Universal Robots PolyScope program: Pallet1.0_PF.urp

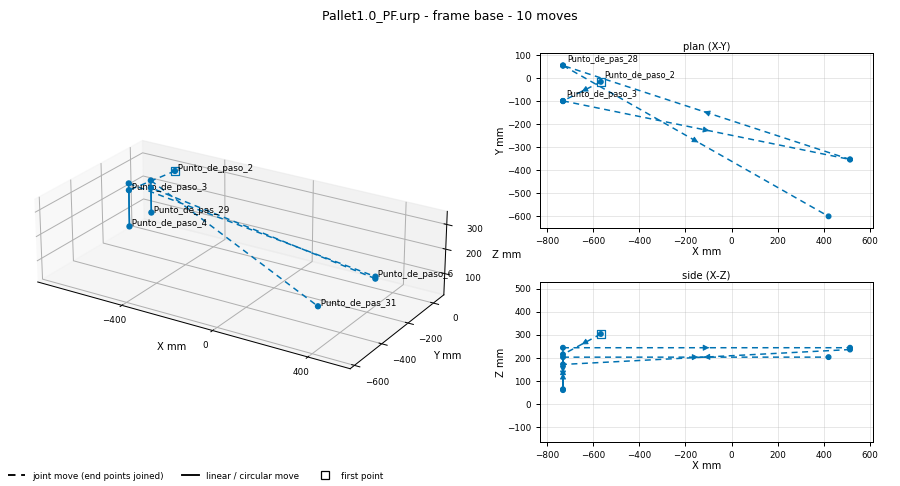
[picture p0: tool path of Pallet1.0_PF.urp in frame base, 10 of 10 moves have a stored position in this frame; points joined in program order, loops and branches not executed]
Program Pallet1.0_PF (installation=default directory=/programs/usbdisk_0 createdIn=3.15.8.106339 lastSavedIn=3.15.8.106339 robotSerialNumber=2015350901)
Calibrated DH parameters: a=[0, -0.425, -0.39225, 0, 0, 0]; d=[0.089159, 0, 0, 0.10915, 0.09465, 0.0823]; alpha=[1.570796, 0, 0, 1.570796, -1.570796, 0]; deltaTheta=[0, 0, 0, 0, 0, 0]
Robot Program (runOnlyOnce=false)
  MoveJ speed 60 deg/s, acceleration 80 deg/s^2 (useActiveTCP=true)
    Waypoint Punto_de_paso_2: TCP in base x=-566.321 y=-16.438 z=304.18 mm, rx=2.2273 ry=2.2091 rz=0.0057 rad; joints [-9.438, -79.943, 72.118, -81.838, -90.015, -8.968] deg; flange x=-567.338 y=-16.315 z=478.176 mm, rx=2.2273 ry=2.2091 rz=0.0057 rad
    If digital_in[1]≟ True
      MoveJ speed 60 deg/s, acceleration 80 deg/s^2 (useActiveTCP=true)
        Waypoint Punto_de_paso_3: TCP in base x=-730.444 y=-98.928 z=215.761 mm, rx=2.2274 ry=2.209 rz=0.0055 rad; joints [-0.817, -54.762, 49.45, -84.36, -89.96, -0.342] deg; flange x=-731.439 y=-98.792 z=389.758 mm, rx=2.2274 ry=2.209 rz=0.0055 rad
        MoveL speed 250 mm/s, acceleration 1200 mm/s^2 (useActiveTCP=true) feature=Base
          Waypoint Punto_de_paso_4: TCP in base x=-730.393 y=-100.609 z=60.935 mm, rx=2.2272 ry=2.209 rz=0.0056 rad; joints [-0.686, -52.453, 68.486, -105.697, -89.955, -0.217] deg; flange x=-731.413 y=-100.461 z=234.932 mm, rx=2.2272 ry=2.209 rz=0.0056 rad
          URCap Gripper (Robotiq_Grippers, Robotiq Inc.) dataModel(position=100.0, force=100.0, speed=100.0, positionInDouble=100.0, forceInDouble=100.0, speedInDouble=100.0, slaveIds=[9], blocking=true); state(isChildrenLocked=true)
          Waypoint Punto_de_paso_5: TCP in base x=-730.487 y=-98.949 z=244.682 mm, rx=2.2273 ry=2.2091 rz=0.0053 rad; joints [-0.817, -54.045, 44.014, -79.647, -89.955, -0.345] deg; flange x=-731.462 y=-98.799 z=418.679 mm, rx=2.2273 ry=2.2091 rz=0.0053 rad
          MoveJ speed 60 deg/s, acceleration 80 deg/s^2 (useActiveTCP=true)
            Waypoint Punto_de_paso_6: TCP in base x=513.312 y=-352.994 z=244.725 mm, rx=2.2039 ry=-2.2386 rz=-0.0089 rad; joints [135.397, -72.477, 71.437, -88.635, -90.007, -43.708] deg; flange x=514.03 y=-353.672 z=418.722 mm, rx=2.2039 ry=-2.2386 rz=-0.0089 rad
          MoveL speed 250 mm/s, acceleration 1200 mm/s^2 (useActiveTCP=true) feature=Base
            Waypoint Punto_de_paso_7: TCP in base x=513.278 y=-353.004 z=236.797 mm, rx=2.2038 ry=-2.2387 rz=-0.0091 rad; joints [135.393, -72.485, 72.603, -89.786, -90.006, -43.706] deg; flange x=514.01 y=-353.701 z=410.794 mm, rx=2.2038 ry=-2.2387 rz=-0.0091 rad
            Pallet pattern(dimensionality=List firstAxisCount=5 secondAxisCount=5 thirdAxisCount=5 motionType=MoveL speed=0.25 acceleration=1.2 useActiveTCP=true, counterVariable(name=cont_1, initializeExpression=0), patternPoseVariable(name=pose_1), feature=Base, children(Waypoint(type=Fixed name=Punto_de_paso_8, position(joints=2.3631303310394287, -1.1275900045977991, 1.6604909896850586, -2.0977628866778772, -1.571042839680807, -0.7629154364215296 pose=0.5132245674611735, -0.3529411145356251, 0.01696247469393014, 2.203863236658737, -2.2383939411612848, -0.009314066402786586), poseInFeatureCoordinates=[0.513225, -0.352941, 0.016962, 2.203863, -2.238394, -0.009314], outputFlangePose=[0.51399, -0.353636, 0.190959, 2.203863, -2.238394, -0.009314]), Waypoint(type=Fixed name=Punto_de_paso_9, position(joints=2.4081342220306396, -1.0566390196429651, 1.545675277709961, -2.05412465730776, -1.570719067250387, -0.7178614775287073 pose=0.5548105961057649, -0.3530178817913074, 0.018104225127487772, 2.2038560559889255, -2.2385008669096638, -0.008956480055837733), poseInFeatureCoordinates=[0.554811, -0.353018, 0.018104, 2.203856, -2.238501, -0.008956], outputFlangePose=[0.555539, -0.353693, 0.192101, 2.203856, -2.238501, -0.008956]), Waypoint(type=Fixed name=Punto_de_pas_10, position(joints=2.446105718612671, -0.9861076513873499, 1.4307241439819336, -2.0095513502704065, -1.5704076925860804, -0.6796610991107386 pose=0.5934753632034022, -0.35301619621523517, 0.017998009023001, 2.203652981289238, -2.2388090833039787, -0.009222219608768033), poseInFeatureCoordinates=[0.593475, -0.353016, 0.017998, 2.203653, -2.238809, -0.009222], outputFlangePose=[0.594215, -0.353722, 0.191995, 2.203653, -2.238809, -0.009222]), Waypoint(type=Fixed name=Punto_de_pas_11, position(joints=2.480747699737549, -0.9116233030902308, 1.3046913146972656, -1.958066765462057, -1.5702398459063929, -0.6444733778582972 pose=0.6321841473893125, -0.35306041061215476, 0.018035419146744114, 2.20302057784513, -2.2393896017985955, -0.009141742887616903), poseInFeatureCoordinates=[0.632184, -0.35306, 0.018035, 2.203021, -2.23939, -0.009142], outputFlangePose=[0.632921, -0.353756, 0.192032, 2.203021, -2.23939, -0.009142]), Waypoint(type=Fixed name=Punto_de_pas_12, position(joints=2.515030860900879, -0.8245127836810511, 1.1525378227233887, -1.892914120350973, -1.570024315510885, -0.6107981840716761 pose=0.6740908514581094, -0.3529593660500304, 0.017973942492954004, 2.2036977466389036, -2.238717787266496, -0.00935099502202368), poseInFeatureCoordinates=[0.674091, -0.352959, 0.017974, 2.203698, -2.238718, -0.009351], outputFlangePose=[0.674845, -0.353671, 0.191971, 2.203698, -2.238718, -0.009351]), Waypoint(type=Fixed name=Punto_de_pas_13, position(joints=2.3630945682525635, -1.169779125844137, 1.6140356063842773, -2.009144131337301, -1.5711506048785608, -0.7630236784564417 pose=0.5131685944157, -0.35295550636586853, 0.05500279295848928, 2.2038697585970315, -2.2382376084810494, -0.00927087314573258), poseInFeatureCoordinates=[0.513169, -0.352956, 0.055003, 2.20387, -2.238238, -0.009271], outputFlangePose=[0.513944, -0.353634, 0.229, 2.20387, -2.238238, -0.009271]), Waypoint(type=Fixed name=Punto_de_pas_14, position(joints=2.4080862998962402, -1.094360653554098, 1.500410556793213, -1.9713957945453089, -1.5707791487323206, -0.7179215590106409 pose=0.5548164047230572, -0.35308568147939057, 0.05508461053102831, 2.20383957497247, -2.23845651633265, -0.008547041026006829), poseInFeatureCoordinates=[0.554816, -0.353086, 0.055085, 2.20384, -2.238457, -0.008547], outputFlangePose=[0.555519, -0.353723, 0.229082, 2.20384, -2.238457, -0.008547]), Waypoint(type=Fixed name=Punto_de_pas_15, position(joints=2.446117877960205, -1.021660629902975, 1.383436679840088, -1.9266999403582972, -1.570467774068014, -0.6796610991107386 pose=0.5934677735696893, -0.35301912054014967, 0.0559910473342225, 2.2036240498734854, -2.238752074764261, -0.00922996533762203), poseInFeatureCoordinates=[0.593468, -0.353019, 0.055991, 2.203624, -2.238752, -0.00923], outputFlangePose=[0.594216, -0.353718, 0.229988, 2.203624, -2.238752, -0.00923]), Waypoint(type=Fixed name=Punto_de_pas_16, position(joints=2.480783700942993, -0.9441817442523401, 1.2555980682373047, -1.8764341513263147, -1.5702040831195276, -0.6444852987872522 pose=0.6321844252540715, -0.3530163761280898, 0.05638557463513269, 2.203100752356905, -2.2393639874148366, -0.009119588993108625), poseInFeatureCoordinates=[0.632184, -0.353016, 0.056386, 2.203101, -2.239364, -0.00912], outputFlangePose=[0.632915, -0.353715, 0.230383, 2.203101, -2.239364, -0.00912]), Waypoint(type=Fixed name=Punto_de_pas_17, position(joints=2.515138626098633, -0.8528311888324183, 1.1003336906433105, -1.8122723738299769, -1.5700843969928187, -0.6107738653766077 pose=0.6741036541561095, -0.35288746982087266, 0.05628562580244548, 2.2037352226759186, -2.238568724907899, -0.009519706762820677), poseInFeatureCoordinates=[0.674104, -0.352887, 0.056286, 2.203735, -2.238569, -0.00952], outputFlangePose=[0.674881, -0.353603, 0.230282, 2.203735, -2.238569, -0.00952]), Waypoint(type=Fixed name=Punto_de_pas_18, position(joints=2.363046646118164, -1.2044346968280237, 1.5590686798095703, -1.9196580092059534, -1.5711386839496058, -0.7629631201373499 pose=0.5131860409950756, -0.3530097003409165, 0.09290491266257156, 2.203758462356244, -2.2383675429672354, -0.009057018848740528), poseInFeatureCoordinates=[0.513186, -0.35301, 0.092905, 2.203758, -2.238368, -0.009057], outputFlangePose=[0.513943, -0.353673, 0.266902, 2.203758, -2.238368, -0.009057]), Waypoint(type=Fixed name=Punto_de_pas_19, position(joints=2.408074378967285, -1.1262005011187952, 1.4451117515563965, -1.8843262831317347, -1.5708149115191858, -0.7178857962237757 pose=0.5548151996713835, -0.3531073422909641, 0.0930535390031054, 2.2037643292926323, -2.2384866218002153, -0.008435196605507001), poseInFeatureCoordinates=[0.554815, -0.353107, 0.093054, 2.203764, -2.238487, -0.008435], outputFlangePose=[0.555513, -0.353732, 0.267051, 2.203764, -2.238487, -0.008435]), Waypoint(type=Fixed name=Punto_de_pas_20, position(joints=2.446141481399536, -1.049763027821676, 1.3284411430358887, -1.8438447157489222, -1.5705392996417444, -0.6796248594867151 pose=0.593499660509277, -0.3530486469996806, 0.09303287538988136, 2.20357754039206, -2.238732576216275, -0.008839450693340935), poseInFeatureCoordinates=[0.5935, -0.353049, 0.093033, 2.203578, -2.238733, -0.008839], outputFlangePose=[0.594223, -0.353711, 0.26703, 2.203578, -2.238733, -0.008839]), Waypoint(type=Fixed name=Punto_de_pas_21, position(joints=2.4808316230773926, -0.9693010489093226, 1.1972637176513672, -1.792868439351217, -1.5702760855304163, -0.6445453802691858 pose=0.6321624175986366, -0.35297919711606884, 0.09406846161006818, 2.20316112021239, -2.2391830633267427, -0.009278826783431064), poseInFeatureCoordinates=[0.632162, -0.352979, 0.094068, 2.203161, -2.239183, -0.009279], outputFlangePose=[0.632916, -0.35368, 0.268065, 2.203161, -2.239183, -0.009279]), Waypoint(type=Fixed name=Punto_de_pas_22, position(joints=2.5151865482330322, -0.8737342993365687, 1.0374155044555664, -1.7285955587970179, -1.570144001637594, -0.6108344236956995 pose=0.674108251554734, -0.3528651117998487, 0.09425003366463722, 2.2038330133524338, -2.2384246855338255, -0.009280286167645216), poseInFeatureCoordinates=[0.674108, -0.352865, 0.09425, 2.203833, -2.238425, -0.00928], outputFlangePose=[0.674871, -0.353557, 0.268247, 2.203833, -2.238425, -0.00928]), Waypoint(type=Fixed name=Punto_de_pas_23, position(joints=2.3629984855651855, -1.2317708174334925, 1.4950027465820312, -1.8283217589007776, -1.571174446736471, -0.7630112806903284 pose=0.5131707080842348, -0.35304893689303485, 0.1310672998062101, 2.2037345545345137, -2.238343056471053, -0.008952794505665341), poseInFeatureCoordinates=[0.513171, -0.353049, 0.131067, 2.203735, -2.238343, -0.008953], outputFlangePose=[0.513924, -0.353699, 0.305064, 2.203735, -2.238343, -0.008953]), Waypoint(type=Fixed name=Punto_de_pas_24, position(joints=2.408074378967285, -1.1507447401629847, 1.3807148933410645, -1.7955272833453577, -1.5708630720721644, -0.7178013960467737 pose=0.554819388099037, -0.35312773426757993, 0.13100770525803954, 2.203642492159454, -2.238551534923004, -0.00820777086849384), poseInFeatureCoordinates=[0.554819, -0.353128, 0.131008, 2.203642, -2.238552, -0.008208], outputFlangePose=[0.555504, -0.353729, 0.305005, 2.203642, -2.238552, -0.008208]), Waypoint(type=Fixed name=Punto_de_pas_25, position(joints=2.445997953414917, -1.0713494459735315, 1.2620959281921387, -1.7558816115008753, -1.5705512205706995, -0.6796129385577601 pose=0.5934510057003118, -0.353139496484484, 0.1310450990567559, 2.2033932515905694, -2.2388933313548534, -0.008886805674271178), poseInFeatureCoordinates=[0.593451, -0.353139, 0.131045, 2.203393, -2.238893, -0.008887], outputFlangePose=[0.59418, -0.353803, 0.305042, 2.203393, -2.238893, -0.008887]), Waypoint(type=Fixed name=Punto_de_pas_26, position(joints=2.480879545211792, -0.9869101683246058, 1.1285271644592285, -1.7065790335284632, -1.5703237692462366, -0.6446173826800745 pose=0.6321941557152236, -0.3529759022987843, 0.13153622061743322, 2.2032678780951342, -2.2390226574753136, -0.009181205365187293), poseInFeatureCoordinates=[0.632194, -0.352976, 0.131536, 2.203268, -2.239023, -0.009181], outputFlangePose=[0.632945, -0.353664, 0.305533, 2.203268, -2.239023, -0.009181]), Waypoint(type=Fixed name=Punto_de_pas_27, position(joints=2.5152344703674316, -0.8862040678607386, 0.9623470306396484, -1.6410678068744105, -1.5702160040484827, -0.6108582655536097 pose=0.6741341209130111, -0.35286206802645803, 0.13170720668516567, 2.203865000162463, -2.238296039311312, -0.009245053414911254), poseInFeatureCoordinates=[0.674134, -0.352862, 0.131707, 2.203865, -2.238296, -0.009245], outputFlangePose=[0.674903, -0.353543, 0.305704, 2.203865, -2.238296, -0.009245]))); actionSequence(name=SecuenciaPalé motionType=MoveL speed=0.25 acceleration=1.2 useActiveTCP=true, anchorWaypoint(type=Fixed name=PuntoDePatrón_1, position(joints=2.3631303310394287, -1.1276257673846644, 1.6605868339538574, -2.097715202962057, -1.5710185209857386, -0.7629755179034632 pose=0.5131909342788984, -0.35289919057667213, 0.01693865784924231, 2.2039461302595416, -2.238343765061751, -0.00948395217768327), poseInFeatureCoordinates=[0.513191, -0.352899, 0.016939, 2.203946, -2.238344, -0.009484], outputFlangePose=[0.513967, -0.35361, 0.190935, 2.203946, -2.238344, -0.009484]), feature=Base, children(Waypoint(type=Fixed name=Acercar_1, position(joints=2.3878726959228516, -1.1627238432513636, 1.499763011932373, -1.901944939290182, -1.5708869139300745, -0.738204304371969 pose=0.535486537471644, -0.35292770718209365, 0.09269323575355731, 2.2039055569885972, -2.238368044698761, -0.009239097655524674), poseInFeatureCoordinates=[0.535487, -0.352928, 0.092693, 2.203906, -2.238368, -0.009239], outputFlangePose=[0.536245, -0.353618, 0.26669, 2.203906, -2.238368, -0.009239]), Waypoint=PuntoDePatrón_1, Contributed(strategyProgramNodeType=Gripper strategyURCapDeveloper=Robotiq Inc. strategyURCapName=Robotiq_Grippers, dataModel(position=0.0, force=100.0, speed=100.0, positionInDouble=0.0, forceInDouble=100.0, speedInDouble=100.0, slaveIds=[9], blocking=true), state(isChildrenLocked=true)), Set(type=NoAction), Wait(type=Sleep, waitTime=1), Waypoint(type=Fixed name=Salir_1, position(joints=2.3556182384490967, -1.2753384749041956, 1.433816909790039, -1.7237561384784144, -1.5711506048785608, -0.7702725569354456 pose=0.5042328769515484, -0.35049239066438986, 0.17702159380140353, 2.2036488263975693, -2.2385225445096353, -0.008663256964435576), poseInFeatureCoordinates=[0.504233, -0.350492, 0.177022, 2.203649, -2.238523, -0.008663], outputFlangePose=[0.504955, -0.351128, 0.351019, 2.203649, -2.238523, -0.008663])))
              Pattern -> pattern
              AnchoredSequence -> SecuenciaPalé
    ElseIf digital_in[0]≟ True
      MoveJ speed 60 deg/s, acceleration 80 deg/s^2 (useActiveTCP=true)
        Waypoint Punto_de_pas_28: TCP in base x=-730.325 y=54.404 z=172.261 mm, rx=2.2271 ry=2.2089 rz=0.0058 rad; joints [-12.82, -55.781, 57.455, -91.329, -90.032, -12.349] deg; flange x=-731.369 y=54.543 z=346.257 mm, rx=2.2271 ry=2.2089 rz=0.0058 rad
        MoveL speed 250 mm/s, acceleration 1200 mm/s^2 (useActiveTCP=true) feature=Base
          Waypoint Punto_de_pas_29: TCP in base x=-730.375 y=54.354 z=64.707 mm, rx=2.2272 ry=2.2093 rz=0.0057 rad; joints [-12.814, -53.288, 69.317, -105.701, -90.036, -12.35] deg; flange x=-731.373 y=54.469 z=238.705 mm, rx=2.2272 ry=2.2093 rz=0.0057 rad
          URCap Gripper (Robotiq_Grippers, Robotiq Inc.) dataModel(position=100.0, force=100.0, speed=100.0, positionInDouble=100.0, forceInDouble=100.0, speedInDouble=100.0, slaveIds=[9], blocking=true); state(isChildrenLocked=true)
          Waypoint Punto_de_pas_30: TCP in base x=-730.317 y=54.385 z=203.798 mm, rx=2.2271 ry=2.209 rz=0.0058 rad; joints [-12.819, -55.724, 52.756, -86.687, -90.032, -12.352] deg; flange x=-731.359 y=54.522 z=377.794 mm, rx=2.2271 ry=2.209 rz=0.0058 rad
          MoveJ speed 60 deg/s, acceleration 80 deg/s^2 (useActiveTCP=true)
            Waypoint Punto_de_pas_31: TCP in base x=420.29 y=-599.707 z=203.949 mm, rx=-2.196 ry=2.245 rz=0.009 rad; joints [116.465, -55.735, 52.753, -86.686, -90.037, -62.27] deg; flange x=420.842 y=-600.562 z=377.946 mm, rx=-2.196 ry=2.245 rz=0.009 rad
            Pallet pattern(dimensionality=List firstAxisCount=5 secondAxisCount=5 thirdAxisCount=5 motionType=MoveL speed=0.25 acceleration=1.2 useActiveTCP=true, counterVariable(name=cont_2, initializeExpression=0), patternPoseVariable(name=pose_2), feature=Base, children(Waypoint(type=Fixed name=Punto_de_pas_32, position(joints=2.0326786041259766, -0.9004228750811976, 1.2612924575805664, -1.9260895887957972, -1.5714500586139124, -1.0868600050555628 pose=0.42031223679203245, -0.5997915862684211, 0.026862123093794543, -2.1960409743045224, 2.245010484936809, 0.008647737661910772), poseInFeatureCoordinates=[0.420312, -0.599792, 0.026862, -2.196041, 2.24501, 0.008648], outputFlangePose=[0.420846, -0.60061, 0.200859, -2.196041, 2.24501, 0.008648]), Waypoint(type=Fixed name=Punto_de_pas_33, position(joints=1.9777237176895142, -0.952315632496969, 1.3581628799438477, -1.9710243383990687, -1.5718210379229944, -1.1419809500323694 pose=0.377052081475406, -0.59975092745355, 0.023745193947307175, -2.1962488525573267, 2.2448477292954836, 0.00881257214877391), poseInFeatureCoordinates=[0.377052, -0.599751, 0.023745, -2.196249, 2.244848, 0.008813], outputFlangePose=[0.377603, -0.600578, 0.197742, -2.196249, 2.244848, 0.008813]), Waypoint(type=Fixed name=Punto_de_pas_34, position(joints=1.9198249578475952, -1.0006139914142054, 1.4385533332824707, -2.0033238569842737, -1.5720370451556605, -1.1997769514666956 pose=0.33410272036293187, -0.5998099590168167, 0.023773719631766138, -2.1961063586547516, 2.24493173781439, 0.0085445244798358), poseInFeatureCoordinates=[0.334103, -0.59981, 0.023774, -2.196106, 2.244932, 0.008545], outputFlangePose=[0.334628, -0.600621, 0.197771, -2.196106, 2.244932, 0.008545]), Waypoint(type=Fixed name=Punto_de_pas_35, position(joints=1.858311414718628, -1.0438936392413538, 1.5088882446289062, -2.030461136494772, -1.5724318663226526, -1.2613032499896448 pose=0.2907433241646436, -0.5997736524692927, 0.02382327555876751, -2.1961600524399834, 2.244955734555862, 0.008598267834922154), poseInFeatureCoordinates=[0.290743, -0.599774, 0.023823, -2.19616, 2.244956, 0.008598], outputFlangePose=[0.291279, -0.600582, 0.197821, -2.19616, 2.244956, 0.008598]), Waypoint(type=Fixed name=Punto_de_pas_36, position(joints=1.7935070991516113, -1.0816510359393519, 1.5690093040466309, -2.0529869238482874, -1.572444264088766, -1.326031510029928 pose=0.2473137524033027, -0.5997893997183813, 0.023847864559044724, -2.195895712983425, 2.2448565162089196, 0.008266422363619219), poseInFeatureCoordinates=[0.247314, -0.599789, 0.023848, -2.195896, 2.244857, 0.008266], outputFlangePose=[0.247792, -0.600603, 0.197845, -2.195896, 2.244857, 0.008266]), Waypoint(type=Fixed name=Punto_de_pas_37, position(joints=2.0326786041259766, -0.9291122595416468, 1.2122488021850586, -1.8483122030841272, -1.5714619795428675, -1.0868719259845179 pose=0.42029785790070623, -0.5997695572523196, 0.06321153303211358, -2.1960526460529084, 2.2449955400753483, 0.00871973716241175), poseInFeatureCoordinates=[0.420298, -0.59977, 0.063212, -2.196053, 2.244996, 0.00872], outputFlangePose=[0.420837, -0.600593, 0.237209, -2.196053, 2.244996, 0.00872]), Waypoint(type=Fixed name=Punto_de_pas_38, position(joints=1.977711796760559, -0.9875810782061976, 1.3046436309814453, -1.8824222723590296, -1.571881119404928, -1.1419933477984827 pose=0.3770293418298652, -0.599758155631741, 0.06479981138223204, -2.196334972325421, 2.244934527389321, 0.008579161455837609), poseInFeatureCoordinates=[0.377029, -0.599758, 0.0648, -2.196335, 2.244935, 0.008579], outputFlangePose=[0.377577, -0.600552, 0.238797, -2.196335, 2.244935, 0.008579]), Waypoint(type=Fixed name=Punto_de_pas_39, position(joints=1.9198849201202393, -1.0374968687640589, 1.3867096900939941, -1.91455585161318, -1.5720132032977503, -1.1998370329486292 pose=0.33413868631545324, -0.5997720606940312, 0.06411739251770301, -2.1962138122624366, 2.2447721167456494, 0.008588305297903552), poseInFeatureCoordinates=[0.334139, -0.599772, 0.064117, -2.196214, 2.244772, 0.008588], outputFlangePose=[0.334662, -0.600591, 0.238115, -2.196214, 2.244772, 0.008588]), Waypoint(type=Fixed name=Punto_de_pas_40, position(joints=1.8583234548568726, -1.0827291647540491, 1.4574856758117676, -1.940078083668844, -1.5723961035357874, -1.2612794081317347 pose=0.29074880148792204, -0.5997319321085388, 0.06414082495110349, -2.1960770296676575, 2.244897320663058, 0.00877291921991509), poseInFeatureCoordinates=[0.290749, -0.599732, 0.064141, -2.196077, 2.244897, 0.008773], outputFlangePose=[0.291286, -0.600566, 0.238138, -2.196077, 2.244897, 0.008773]), Waypoint(type=Fixed name=Punto_de_pas_41, position(joints=1.793459177017212, -1.122235123311178, 1.5176410675048828, -1.9610002676593226, -1.5724080244647425, -1.326019589100973 pose=0.24729580851692193, -0.599806887646094, 0.06423806217654832, -2.195794209303443, 2.244887267137956, 0.008282342822273286), poseInFeatureCoordinates=[0.247296, -0.599807, 0.064238, -2.195794, 2.244887, 0.008282], outputFlangePose=[0.247769, -0.600628, 0.238235, -2.195794, 2.244887, 0.008282]), Waypoint(type=Fixed name=Punto_de_pas_42, position(joints=2.0327625274658203, -0.954195801411764, 1.1431756019592285, -1.7539165655719202, -1.5714500586139124, -1.0869205633746546 pose=0.4203303793998149, -0.5996916537066742, 0.10535776894644641, -2.1961415723694313, 2.244788685731963, 0.009070726951884931), poseInFeatureCoordinates=[0.42033, -0.599692, 0.105358, -2.196142, 2.244789, 0.009071], outputFlangePose=[0.420887, -0.600554, 0.279355, -2.196142, 2.244789, 0.009071]), Waypoint(type=Fixed name=Punto_de_pas_43, position(joints=1.9777237176895142, -1.0141261259662073, 1.2409725189208984, -1.792258087788717, -1.5719292799579065, -1.1419933477984827 pose=0.37703210936377796, -0.5997746804500261, 0.10496705431930384, -2.196393074106652, 2.2449669183053333, 0.008530349931466608), poseInFeatureCoordinates=[0.377032, -0.599775, 0.104967, -2.196393, 2.244967, 0.00853], outputFlangePose=[0.377584, -0.600557, 0.278964, -2.196393, 2.244967, 0.00853]), Waypoint(type=Fixed name=Punto_de_pas_44, position(joints=1.9198368787765503, -1.0666535536395472, 1.3238019943237305, -1.8223932425128382, -1.572000805531637, -1.1998127142535608 pose=0.33410991599099243, -0.5997789419527765, 0.10470445516853558, -2.196096078503044, 2.244814190905074, 0.008720600650474676), poseInFeatureCoordinates=[0.33411, -0.599779, 0.104704, -2.196096, 2.244814, 0.008721], outputFlangePose=[0.334637, -0.600615, 0.278702, -2.196096, 2.244814, 0.008721]), Waypoint(type=Fixed name=Punto_de_pas_45, position(joints=1.8582634925842285, -1.1132872740374964, 1.3967084884643555, -1.8485992590533655, -1.5723722616778772, -1.2612674872027796 pose=0.29071172575896925, -0.5997240448407468, 0.103933136884969, -2.195934251159368, 2.244912665537146, 0.008954286941669805), poseInFeatureCoordinates=[0.290712, -0.599724, 0.103933, -2.195934, 2.244913, 0.008954], outputFlangePose=[0.291252, -0.600584, 0.27793, -2.195934, 2.244913, 0.008954]), Waypoint(type=Fixed name=Punto_de_pas_46, position(joints=1.7934471368789673, -1.1543868223773401, 1.4572100639343262, -1.8684333006488245, -1.572444264088766, -1.326043430958883 pose=0.24728308642957084, -0.5998276339892976, 0.10407914707263485, -2.195834812915026, 2.244902095677252, 0.008291189682723576), poseInFeatureCoordinates=[0.247283, -0.599828, 0.104079, -2.195835, 2.244902, 0.008291], outputFlangePose=[0.247762, -0.600644, 0.278077, -2.195835, 2.244902, 0.008291]), Waypoint(type=Fixed name=Punto_de_pas_47, position(joints=2.0327625274658203, -0.9690373579608362, 1.0653080940246582, -1.6610124746905726, -1.5714381376849573, -1.0869563261615198 pose=0.4203081983806019, -0.5996402495488459, 0.14493178311690272, -2.1961312218118367, 2.2446977464728315, 0.009356126142767485), poseInFeatureCoordinates=[0.420308, -0.59964, 0.144932, -2.196131, 2.244698, 0.009356], outputFlangePose=[0.420878, -0.600534, 0.318929, -2.196131, 2.244698, 0.009356]), Waypoint(type=Fixed name=Punto_de_pas_48, position(joints=1.9776397943496704, -1.0324056784259241, 1.16448974609375, -1.6974156538592737, -1.5719412008868616, -1.1420052687274378 pose=0.3769706546307442, -0.5997882376839357, 0.14556367402348097, -2.196299567358495, 2.245032849351386, 0.008654356965162757), poseInFeatureCoordinates=[0.376971, -0.599788, 0.145564, -2.1963, 2.245033, 0.008654], outputFlangePose=[0.37753, -0.600583, 0.319561, -2.1963, 2.245033, 0.008654]), Waypoint(type=Fixed name=Punto_de_pas_49, position(joints=1.9197770357131958, -1.087029759083883, 1.2509584426879883, -1.7291463057147425, -1.571988884602682, -1.1999085585223597 pose=0.3340794065402006, -0.5998047954020302, 0.14455268321738438, -2.196120666175572, 2.244758527047815, 0.008751538844001079), poseInFeatureCoordinates=[0.334079, -0.599805, 0.144553, -2.196121, 2.244759, 0.008752], outputFlangePose=[0.334606, -0.600646, 0.31855, -2.196121, 2.244759, 0.008752]), Waypoint(type=Fixed name=Punto_de_pas_50, position(joints=1.8582993745803833, -1.1360352675067347, 1.3243889808654785, -1.7533896605121058, -1.5723722616778772, -1.261207405720846 pose=0.2907201279675694, -0.5996692536232531, 0.14433523831004902, -2.1958605212249998, 2.244891377498346, 0.009151380483949976), poseInFeatureCoordinates=[0.29072, -0.599669, 0.144335, -2.195861, 2.244891, 0.009151], outputFlangePose=[0.291267, -0.600553, 0.318332, -2.195861, 2.244891, 0.009151]), Waypoint(type=Fixed name=Punto_de_pas_51, position(joints=1.793339729309082, -1.178033177052633, 1.3882684707641602, -1.7758844534503382, -1.5724080244647425, -1.326031510029928 pose=0.24722403435648985, -0.5998358617025912, 0.14315527141451476, -2.1956934541638375, 2.2450258052720597, 0.008208954346305801), poseInFeatureCoordinates=[0.247224, -0.599836, 0.143155, -2.195693, 2.245026, 0.008209], outputFlangePose=[0.247695, -0.600647, 0.317153, -2.195693, 2.245026, 0.008209]))); actionSequence(name=SecuenciaPalé motionType=MoveL speed=0.25 acceleration=1.2 useActiveTCP=true, anchorWaypoint(type=Fixed name=PuntoDePatrón_2, position(joints=2.0326905250549316, -0.9004471937762659, 1.2612686157226562, -1.9260175863849085, -1.5713780562030237, -1.0868719259845179 pose=0.4203325415800726, -0.5997715907783921, 0.026883984710863146, -2.1960144812733886, 2.2449302994155764, 0.008648395330919075), poseInFeatureCoordinates=[0.420333, -0.599772, 0.026884, -2.196014, 2.24493, 0.008648], outputFlangePose=[0.420857, -0.600599, 0.200881, -2.196014, 2.24493, 0.008648]), feature=Base, children(Waypoint(type=Fixed name=Acercar_2, position(joints=2.032750368118286, -0.951153580342428, 1.1540484428405762, -1.7680748144732874, -1.5714262167560022, -1.086883846913473 pose=0.42035242239054144, -0.599741973292872, 0.09927745608604205, -2.196123752652395, 2.244880544160503, 0.008696023418901055), poseInFeatureCoordinates=[0.420352, -0.599742, 0.099277, -2.196124, 2.244881, 0.008696], outputFlangePose=[0.420886, -0.600568, 0.273275, -2.196124, 2.244881, 0.008696]), Waypoint=PuntoDePatrón_2, Contributed(strategyProgramNodeType=Gripper strategyURCapDeveloper=Robotiq Inc. strategyURCapName=Robotiq_Grippers, dataModel(position=0.0, force=100.0, speed=100.0, positionInDouble=0.0, forceInDouble=100.0, speedInDouble=100.0, slaveIds=[9], blocking=true), state(isChildrenLocked=true)), Set(type=NoAction), Wait(type=Sleep, waitTime=1), Waypoint(type=Fixed name=Salir_2, position(joints=1.950283169746399, -1.0369694868670862, 1.291839599609375, -1.8202012220965784, -1.5718453566180628, -1.1694629828082483 pose=0.35640023268911075, -0.599720957580411, 0.09931984744575259, -2.196245557973125, 2.244751242458276, 0.008554699001879149), poseInFeatureCoordinates=[0.3564, -0.599721, 0.09932, -2.196246, 2.244751, 0.008555], outputFlangePose=[0.356922, -0.600537, 0.273317, -2.196246, 2.244751, 0.008555])))
              Pattern -> pattern
              AnchoredSequence -> SecuenciaPalé
